(* IEC 61131-3 sources: HappyLearnCodesys/content/softmotion/CNC15_LargeGCode, 3 files *)

(* ---- GVL_PARAMETERS.st ---- *)
VAR_GLOBAL
	piMaxDifference : SMC_PosInfo := (dX:= 0.1, dY:= 0.1, dZ:= 0.1, dA := 0.04, dB := 0.04, dC := 0.04);
	dAngleTol : LREAL := 0.01;
	dMinCurvatureRadius : LREAL := 0.015;

	dwTaskCycleMicros : DWORD := 4000;
	dJerkMax : LREAL := 10000;
END_VAR

(* ---- Control.st ---- *)
PROGRAM Control
VAR
	pow1, pow2 : MC_Power := (Enable:= TRUE, bRegulatorOn:= TRUE, bDriveStart:= TRUE);
	cap1, cap2 : SMC_ControlAxisByPos := (bAvoidGaps:= FALSE);
	ipo : SMC_Interpolator := (
		iVelMode:= SMC_INT_VELMODE.QUADRATIC,
		dwIpoTime:= dwTaskCycleMicros,
		dJerkMax:= dJerkMax);

	bInitialized : BOOL;
END_VAR

pow1(Axis := Drive1);
pow2(Axis := Drive2);

IF NOT bInitialized THEN
	IF pow1.Status AND pow2.Status THEN
		bInitialized := TRUE;
	END_IF
END_IF

ipo(bExecute:= bInitialized, poqDataIn := Path.poqDataOut);

cap1(Axis := Drive1,
     iStatus := ipo.iStatus,
	 bEnable := ipo.bWorking,
	 fSetPosition := ipo.piSetPosition.dX);

cap2(Axis := Drive2,
     iStatus := ipo.iStatus,
	 bEnable := ipo.bWorking,
	 fSetPosition := ipo.piSetPosition.dY);

(* ---- Path.st ---- *)
PROGRAM Path
VAR_OUTPUT
	poqDataOut : POINTER TO SMC_OUTQUEUE;
END_VAR
VAR
	rncf : SMC_ReadNCFile2;
	ip : SMC_NCInterpreter;
	smm : SMC_SmoothMerge;
	smp : SMC_SmoothPath;

	cv : SMC_CheckVelocities;

	aBufIp : ARRAY[0..130] OF SMC_GeoInfo;
	aBufSmm  : ARRAY[0..15] OF SMC_GeoInfo;
	aBufSmp : ARRAY[0..99] OF SMC_GeoInfo;
END_VAR
VAR_TEMP
	counter : DINT;
END_VAR

// Set this value depending on your other tasks, PLC performance, and G-Code
counter := 25;

WHILE counter > 0 AND
      (poqDataOut = 0 OR_ELSE (NOT poqDataOut^.bFull AND NOT poqDataOut^.bEndOfList))
DO
	rncf(
		bExecute:= TRUE,
		sFileName:= '_cnc/CNC.cnc');

	ip(
		sentences:= rncf.sentences,
		bExecute:= rncf.bExecute,
		nSizeOutQueue:= SIZEOF(aBufIp),
		pbyBufferOutQueue:= ADR(aBufIp));

	smm(
		bExecute:= ip.bExecute,
		poqDataIn:= ip.poqDataOut,
		nSizeOutQueue:= SIZEOF(aBufSmm),
		pbyBufferOutQueue:= ADR(aBufSmm),
		piMaxDifference:= piMaxDifference,
        usiMaxDegree:= 5,
        wFeatureFlag:= 1,
		dMinimumCurvatureRadius:= dMinCurvatureRadius);

	smp(
		bExecute:= ip.bExecute,
		poqDataIn:= smm.poqDataOut,
		eMode:= SMC_SMOOTHPATHMODE.SP_SPLINE5_MIN_CURVATURE,
		eAddAxMode:= SMC_SMOOTHPATHADDAXMODE.SPAA_EXACT,
		nSizeOutQueue:= SIZEOF(aBufSmp),
		pbyBufferOutQueue:= ADR(aBufSmp),
		dAngleTol:= dAngleTol,
		bSymmetricalDistances:= TRUE,
		bImprovedSymmetricCuts:= TRUE);

	cv(
		bExecute:= ip.bExecute,
		poqDataIn:= smp.poqDataOut,
		dAngleTol:= dAngleTol);

	counter := counter - 1;
END_WHILE

poqDataOut := cv.poqDataOut;
